VAR_GLOBAL
	fbPayloadCarrier : PayloadCarrier;
END_VAR

(* stored: Version 1.1.0.1, ProductVersion 3.1.4024.2
   GVL Global: Id {e05dedbf-06be-4664-9b7f-45382800bf03} *)
